(* CODESYS project Joint_7_TCP_new.project

Project tree, tasks and I/O mapping:
  Device : CODESYS Control arm CTH3 C37-000S1, 3S - Smart Software Solutions GmbH, version 3.5.4.30
    application Application
      libraries: Standard, * (System); Co-Trust Modbus Library, 1.1 (Co-Trust)
      task MainTask (cyclic, interval t#20ms, priority 1) calls Cyclic, TCP
      task EtherCAT_Master (cyclic, interval 2000 µs, priority 0) calls EtherCAT_Master.EtherCAT_Task [EtherCAT_Master.EtherCAT_Task], PLC_PRG
      program PLC_PRG [LD]
      global variables GVL
      trace Trace (task EtherCAT_Master): x.fSetPosition
      function block String_TO_HMI [ST]
      program Cyclic [LD]
      global variables PersistentVars
      program TCP [LD]
    SoftMotion General Axis Pool
    Co-trust LocalBus
    EtherCAT_Master : EtherCAT Master, 3S - Smart Software Solutions GmbH, version 3.5.4.0
        settings: MasterCycleTime = 2000; SlaveAutoRestart = True; NetworkName = 'eth1'; SelectNetworkByName = True; SrcAddress1 = 96; SrcAddress2 = 1856707308
      CiA402_Motor_Control_Device_6 : SOMANET CiA402 Drive, Synapticon GmbH, version Revision=16#0A000002
          settings: Number of Outputs = 7; Number of Inputs = 5; Number of Infos about Outputs = 7; Number of Infos about Inputs = 5; EnableExpertSettings = True; CheckProductID = False; CheckVendorID = False; Sync.Length = 19; Sync.Length = 13; FMMU.Length = 19; FMMU.Length = 13; DC enable = 1; DC sync0 enable = 1; DC sync0 shift time = 0; DC sync1 enable = 0; DC sync1 shift time = 0; DCSetting = 1; RxTxPdo.Sm = -1; RxTxPdo.Sm = -1; RxTxPdo.Sm = -1; RxTxPdo.Sm = -1; RxTxPdo.Sm = -1
          unmapped channels: Controlword, Op Mode, Target Torque, Target Position, Target Velocity, Torque offset, Tuning command, Statusword, Op Mode Display, Position Value, Velocity Value, Torque Value
        Joint_6 : SM_Drive_GenericDSP402, 3S - Smart Software Solutions GmbH, order no. 0, version 3.5.4.10
            settings: dwRatioTechUnitsDenom = 26214400; ScalingIncs = 262144; ScalingMotorTurns2 = 100; AdrOffset_8010 = 120; BitOffset_8010 = 0; BitLength_8010 = 16; Address_8010 = '%QW60'; Type_8010 = 'UINT'; AddressPointer_8010 = ADR(%QW60); AdrOffset_8020 = 128; BitOffset_8020 = 0; BitLength_8020 = 32; Address_8020 = '%QD32'; Type_8020 = 'DINT'; AddressPointer_8020 = ADR(%QD32); AdrOffset_8030 = 132; BitOffset_8030 = 0; BitLength_8030 = 32; Address_8030 = '%QD33'; Type_8030 = 'DINT'; AddressPointer_8030 = ADR(%QD33); AdrOffset_8040 = 124; BitOffset_8040 = 0; BitLength_8040 = 16; Address_8040 = '%QW62'; Type_8040 = 'INT'; AddressPointer_8040 = ADR(%QW62); AdrOffset_8050 = 122; BitOffset_8050 = 0; BitLength_8050 = 8; Address_8050 = '%QB122'; Type_8050 = 'SINT'; AddressPointer_8050 = ADR(%QB122); AdrOffset_8060 = 16#FFFFFFFF; BitOffset_8060 = 0; BitLength_8060 = 0; Address_8060 = ''; Type_8060 = ''; AddressPointer_8060 = 0; AdrOffset_8070 = 16#FFFFFFFF;
              BitOffset_8070 = 0; BitLength_8070 = 0; Address_8070 = ''; Type_8070 = ''; AddressPointer_8070 = 0; AdrOffset_8080 = 136; BitOffset_8080 = 0; BitLength_8080 = 16; Address_8080 = '%QW68'; Type_8080 = 'INT'; AddressPointer_8080 = ADR(%QW68); AdrOffset_8510 = 80; BitOffset_8510 = 0; BitLength_8510 = 16; Address_8510 = '%IW40'; Type_8510 = 'UINT'; AddressPointer_8510 = ADR(%IW40); AdrOffset_8520 = 84; BitOffset_8520 = 0; BitLength_8520 = 32; Address_8520 = '%ID21'; Type_8520 = 'DINT'; AddressPointer_8520 = ADR(%ID21); AdrOffset_8530 = 88; BitOffset_8530 = 0; BitLength_8530 = 32; Address_8530 = '%ID22'; Type_8530 = 'DINT'; AddressPointer_8530 = ADR(%ID22); AdrOffset_8540 = 92; BitOffset_8540 = 0; BitLength_8540 = 16; Address_8540 = '%IW46'; Type_8540 = 'INT'; AddressPointer_8540 = ADR(%IW46); AdrOffset_8550 = 82; BitOffset_8550 = 0; BitLength_8550 = 8; Address_8550 = '%IB82'; Type_8550 = 'SINT';
              AddressPointer_8550 = ADR(%IB82); AdrOffset_8560 = 16#FFFFFFFF; BitOffset_8560 = 0; BitLength_8560 = 0; Address_8560 = ''; Type_8560 = ''; AddressPointer_8560 = 0; AdrOffset_8570 = 16#FFFFFFFF; BitOffset_8570 = 0; BitLength_8570 = 0; Address_8570 = ''; Type_8570 = ''; AddressPointer_8570 = 0; AdrOffset_8580 = 16#FFFFFFFF; BitOffset_8580 = 0; BitLength_8580 = 0; Address_8580 = ''; Type_8580 = ''; AddressPointer_8580 = 0; AdrOffset_8590 = 16#FFFFFFFF; BitOffset_8590 = 0; BitLength_8590 = 0; Address_8590 = ''; Type_8590 = ''; AddressPointer_8590 = 0; AdrOffset_8600 = 16#FFFFFFFF; BitOffset_8600 = 0; BitLength_8600 = 0; Address_8600 = ''; Type_8600 = ''; AddressPointer_8600 = 0; AdrOffset_8600 = 16#FFFFFFFF; BitOffset_8600 = 0; BitLength_8600 = 0; Address_8610 = ''; Type_8610 = ''; AddressPointer_8610 = 0
      CiA402_Motor_Control_Device_4 : SOMANET CiA402 Drive, Synapticon GmbH, version Revision=16#0A000002
          settings: Number of Outputs = 7; Number of Inputs = 5; Number of Infos about Outputs = 7; Number of Infos about Inputs = 5; EnableExpertSettings = True; CheckProductID = False; CheckVendorID = False; Sync.Length = 19; Sync.Length = 13; FMMU.Length = 19; FMMU.Length = 13; DC enable = 1; DC sync0 enable = 1; DC sync0 shift time = 0; DC sync1 enable = 0; DC sync1 shift time = 0; DCSetting = 1; RxTxPdo.Sm = -1; RxTxPdo.Sm = -1; RxTxPdo.Sm = -1; RxTxPdo.Sm = -1; RxTxPdo.Sm = -1
          unmapped channels: Controlword, Op Mode, Target Torque, Target Position, Target Velocity, Torque offset, Tuning command, Statusword, Op Mode Display, Position Value, Velocity Value, Torque Value
        Joint_4 : SM_Drive_GenericDSP402, 3S - Smart Software Solutions GmbH, order no. 0, version 3.5.4.10
            settings: dwRatioTechUnitsDenom = 26214400; fSWLimitDeceleration = 0.0; fSWErrorMaxDistance = 0.0; ScalingIncs = 262144; ScalingMotorTurns2 = 100; AdrOffset_8010 = 72; BitOffset_8010 = 0; BitLength_8010 = 16; Address_8010 = '%QW36'; Type_8010 = 'UINT'; AddressPointer_8010 = ADR(%QW36); AdrOffset_8020 = 80; BitOffset_8020 = 0; BitLength_8020 = 32; Address_8020 = '%QD20'; Type_8020 = 'DINT'; AddressPointer_8020 = ADR(%QD20); AdrOffset_8030 = 84; BitOffset_8030 = 0; BitLength_8030 = 32; Address_8030 = '%QD21'; Type_8030 = 'DINT'; AddressPointer_8030 = ADR(%QD21); AdrOffset_8040 = 76; BitOffset_8040 = 0; BitLength_8040 = 16; Address_8040 = '%QW38'; Type_8040 = 'INT'; AddressPointer_8040 = ADR(%QW38); AdrOffset_8050 = 74; BitOffset_8050 = 0; BitLength_8050 = 8; Address_8050 = '%QB74'; Type_8050 = 'SINT'; AddressPointer_8050 = ADR(%QB74); AdrOffset_8060 = 16#FFFFFFFF; BitOffset_8060 = 0; BitLength_8060 = 0; Address_8060 = ''; Type_8060 = '';
              AddressPointer_8060 = 0; AdrOffset_8070 = 16#FFFFFFFF; BitOffset_8070 = 0; BitLength_8070 = 0; Address_8070 = ''; Type_8070 = ''; AddressPointer_8070 = 0; AdrOffset_8080 = 88; BitOffset_8080 = 0; BitLength_8080 = 16; Address_8080 = '%QW44'; Type_8080 = 'INT'; AddressPointer_8080 = ADR(%QW44); AdrOffset_8510 = 48; BitOffset_8510 = 0; BitLength_8510 = 16; Address_8510 = '%IW24'; Type_8510 = 'UINT'; AddressPointer_8510 = ADR(%IW24); AdrOffset_8520 = 52; BitOffset_8520 = 0; BitLength_8520 = 32; Address_8520 = '%ID13'; Type_8520 = 'DINT'; AddressPointer_8520 = ADR(%ID13); AdrOffset_8530 = 56; BitOffset_8530 = 0; BitLength_8530 = 32; Address_8530 = '%ID14'; Type_8530 = 'DINT'; AddressPointer_8530 = ADR(%ID14); AdrOffset_8540 = 60; BitOffset_8540 = 0; BitLength_8540 = 16; Address_8540 = '%IW30'; Type_8540 = 'INT'; AddressPointer_8540 = ADR(%IW30); AdrOffset_8550 = 50; BitOffset_8550 = 0; BitLength_8550 = 8;
              Address_8550 = '%IB50'; Type_8550 = 'SINT'; AddressPointer_8550 = ADR(%IB50); AdrOffset_8560 = 16#FFFFFFFF; BitOffset_8560 = 0; BitLength_8560 = 0; Address_8560 = ''; Type_8560 = ''; AddressPointer_8560 = 0; AdrOffset_8570 = 16#FFFFFFFF; BitOffset_8570 = 0; BitLength_8570 = 0; Address_8570 = ''; Type_8570 = ''; AddressPointer_8570 = 0; AdrOffset_8580 = 16#FFFFFFFF; BitOffset_8580 = 0; BitLength_8580 = 0; Address_8580 = ''; Type_8580 = ''; AddressPointer_8580 = 0; AdrOffset_8590 = 16#FFFFFFFF; BitOffset_8590 = 0; BitLength_8590 = 0; Address_8590 = ''; Type_8590 = ''; AddressPointer_8590 = 0; AdrOffset_8600 = 16#FFFFFFFF; BitOffset_8600 = 0; BitLength_8600 = 0; Address_8600 = ''; Type_8600 = ''; AddressPointer_8600 = 0; AdrOffset_8600 = 16#FFFFFFFF; BitOffset_8600 = 0; BitLength_8600 = 0; Address_8610 = ''; Type_8610 = ''; AddressPointer_8610 = 0
      CiA402_Motor_Control_Device_2 : SOMANET CiA402 Drive, Synapticon GmbH, version Revision=16#0A000002
          settings: Number of Outputs = 7; Number of Inputs = 5; Number of Infos about Outputs = 7; Number of Infos about Inputs = 5; EnableExpertSettings = True; CheckProductID = False; CheckVendorID = False; Sync.Length = 19; Sync.Length = 13; FMMU.Length = 19; FMMU.Length = 13; DC enable = 1; DC sync0 enable = 1; DC sync0 shift time = 0; DC sync1 enable = 0; DC sync1 shift time = 0; DCSetting = 1; RxTxPdo.Sm = -1; RxTxPdo.Sm = -1; RxTxPdo.Sm = -1; RxTxPdo.Sm = -1; RxTxPdo.Sm = -1
          unmapped channels: Controlword, Op Mode, Target Torque, Target Position, Target Velocity, Torque offset, Tuning command, Statusword, Op Mode Display, Position Value, Velocity Value, Torque Value
        Joint_2 : SM_Drive_GenericDSP402, 3S - Smart Software Solutions GmbH, order no. 0, version 3.5.4.10
            settings: dwRatioTechUnitsDenom = 31457280; ScalingIncs = 262144; ScalingMotorTurns2 = 120; AdrOffset_8010 = 24; BitOffset_8010 = 0; BitLength_8010 = 16; Address_8010 = '%QW12'; Type_8010 = 'UINT'; AddressPointer_8010 = ADR(%QW12); AdrOffset_8020 = 32; BitOffset_8020 = 0; BitLength_8020 = 32; Address_8020 = '%QD8'; Type_8020 = 'DINT'; AddressPointer_8020 = ADR(%QD8); AdrOffset_8030 = 36; BitOffset_8030 = 0; BitLength_8030 = 32; Address_8030 = '%QD9'; Type_8030 = 'DINT'; AddressPointer_8030 = ADR(%QD9); AdrOffset_8040 = 28; BitOffset_8040 = 0; BitLength_8040 = 16; Address_8040 = '%QW14'; Type_8040 = 'INT'; AddressPointer_8040 = ADR(%QW14); AdrOffset_8050 = 26; BitOffset_8050 = 0; BitLength_8050 = 8; Address_8050 = '%QB26'; Type_8050 = 'SINT'; AddressPointer_8050 = ADR(%QB26); AdrOffset_8060 = 16#FFFFFFFF; BitOffset_8060 = 0; BitLength_8060 = 0; Address_8060 = ''; Type_8060 = ''; AddressPointer_8060 = 0; AdrOffset_8070 = 16#FFFFFFFF;
              BitOffset_8070 = 0; BitLength_8070 = 0; Address_8070 = ''; Type_8070 = ''; AddressPointer_8070 = 0; AdrOffset_8080 = 40; BitOffset_8080 = 0; BitLength_8080 = 16; Address_8080 = '%QW20'; Type_8080 = 'INT'; AddressPointer_8080 = ADR(%QW20); AdrOffset_8510 = 16; BitOffset_8510 = 0; BitLength_8510 = 16; Address_8510 = '%IW8'; Type_8510 = 'UINT'; AddressPointer_8510 = ADR(%IW8); AdrOffset_8520 = 20; BitOffset_8520 = 0; BitLength_8520 = 32; Address_8520 = '%ID5'; Type_8520 = 'DINT'; AddressPointer_8520 = ADR(%ID5); AdrOffset_8530 = 24; BitOffset_8530 = 0; BitLength_8530 = 32; Address_8530 = '%ID6'; Type_8530 = 'DINT'; AddressPointer_8530 = ADR(%ID6); AdrOffset_8540 = 28; BitOffset_8540 = 0; BitLength_8540 = 16; Address_8540 = '%IW14'; Type_8540 = 'INT'; AddressPointer_8540 = ADR(%IW14); AdrOffset_8550 = 18; BitOffset_8550 = 0; BitLength_8550 = 8; Address_8550 = '%IB18'; Type_8550 = 'SINT';
              AddressPointer_8550 = ADR(%IB18); AdrOffset_8560 = 16#FFFFFFFF; BitOffset_8560 = 0; BitLength_8560 = 0; Address_8560 = ''; Type_8560 = ''; AddressPointer_8560 = 0; AdrOffset_8570 = 16#FFFFFFFF; BitOffset_8570 = 0; BitLength_8570 = 0; Address_8570 = ''; Type_8570 = ''; AddressPointer_8570 = 0; AdrOffset_8580 = 16#FFFFFFFF; BitOffset_8580 = 0; BitLength_8580 = 0; Address_8580 = ''; Type_8580 = ''; AddressPointer_8580 = 0; AdrOffset_8590 = 16#FFFFFFFF; BitOffset_8590 = 0; BitLength_8590 = 0; Address_8590 = ''; Type_8590 = ''; AddressPointer_8590 = 0; AdrOffset_8600 = 16#FFFFFFFF; BitOffset_8600 = 0; BitLength_8600 = 0; Address_8600 = ''; Type_8600 = ''; AddressPointer_8600 = 0; AdrOffset_8600 = 16#FFFFFFFF; BitOffset_8600 = 0; BitLength_8600 = 0; Address_8610 = ''; Type_8610 = ''; AddressPointer_8610 = 0
      CiA402_Motor_Control_Device : SOMANET CiA402 Drive, Synapticon GmbH, version Revision=16#0A000002
          settings: Number of Outputs = 7; Number of Inputs = 5; Number of Infos about Outputs = 7; Number of Infos about Inputs = 5; EnableExpertSettings = True; CheckProductID = False; CheckVendorID = False; Sync.Length = 19; Sync.Length = 13; FMMU.Length = 19; FMMU.Length = 13; DC enable = 1; DC sync0 enable = 1; DC sync0 shift time = 0; DC sync1 enable = 0; DC sync1 shift time = 0; DCSetting = 1; RxTxPdo.Sm = -1; RxTxPdo.Sm = -1; RxTxPdo.Sm = -1; RxTxPdo.Sm = -1; RxTxPdo.Sm = -1
          unmapped channels: Controlword, Op Mode, Target Torque, Target Position, Target Velocity, Torque offset, Tuning command, Statusword, Op Mode Display, Position Value, Velocity Value, Torque Value
        Joint_7 : SM_Drive_GenericDSP402, 3S - Smart Software Solutions GmbH, order no. 0, version 3.5.4.10
            settings: dwRatioTechUnitsDenom = 26214400; ScalingIncs = 262144; ScalingMotorTurns2 = 100; AdrOffset_8010 = 144; BitOffset_8010 = 0; BitLength_8010 = 16; Address_8010 = '%QW72'; Type_8010 = 'UINT'; AddressPointer_8010 = ADR(%QW72); AdrOffset_8020 = 152; BitOffset_8020 = 0; BitLength_8020 = 32; Address_8020 = '%QD38'; Type_8020 = 'DINT'; AddressPointer_8020 = ADR(%QD38); AdrOffset_8030 = 156; BitOffset_8030 = 0; BitLength_8030 = 32; Address_8030 = '%QD39'; Type_8030 = 'DINT'; AddressPointer_8030 = ADR(%QD39); AdrOffset_8040 = 148; BitOffset_8040 = 0; BitLength_8040 = 16; Address_8040 = '%QW74'; Type_8040 = 'INT'; AddressPointer_8040 = ADR(%QW74); AdrOffset_8050 = 146; BitOffset_8050 = 0; BitLength_8050 = 8; Address_8050 = '%QB146'; Type_8050 = 'SINT'; AddressPointer_8050 = ADR(%QB146); AdrOffset_8060 = 16#FFFFFFFF; BitOffset_8060 = 0; BitLength_8060 = 0; Address_8060 = ''; Type_8060 = ''; AddressPointer_8060 = 0; AdrOffset_8070 = 176;
              BitOffset_8070 = 0; BitLength_8070 = 32; Address_8070 = '%QD44'; Type_8070 = 'DINT'; AddressPointer_8070 = ADR(%QD44); AdrOffset_8080 = 160; BitOffset_8080 = 0; BitLength_8080 = 16; Address_8080 = '%QW80'; Type_8080 = 'INT'; AddressPointer_8080 = ADR(%QW80); AdrOffset_8510 = 96; BitOffset_8510 = 0; BitLength_8510 = 16; Address_8510 = '%IW48'; Type_8510 = 'UINT'; AddressPointer_8510 = ADR(%IW48); AdrOffset_8520 = 100; BitOffset_8520 = 0; BitLength_8520 = 32; Address_8520 = '%ID25'; Type_8520 = 'DINT'; AddressPointer_8520 = ADR(%ID25); AdrOffset_8530 = 104; BitOffset_8530 = 0; BitLength_8530 = 32; Address_8530 = '%ID26'; Type_8530 = 'DINT'; AddressPointer_8530 = ADR(%ID26); AdrOffset_8540 = 108; BitOffset_8540 = 0; BitLength_8540 = 16; Address_8540 = '%IW54'; Type_8540 = 'INT'; AddressPointer_8540 = ADR(%IW54); AdrOffset_8550 = 98; BitOffset_8550 = 0; BitLength_8550 = 8; Address_8550 = '%IB98'; Type_8550 = 'SINT';
              AddressPointer_8550 = ADR(%IB98); AdrOffset_8560 = 16#FFFFFFFF; BitOffset_8560 = 0; BitLength_8560 = 0; Address_8560 = ''; Type_8560 = ''; AddressPointer_8560 = 0; AdrOffset_8570 = 16#FFFFFFFF; BitOffset_8570 = 0; BitLength_8570 = 0; Address_8570 = ''; Type_8570 = ''; AddressPointer_8570 = 0; AdrOffset_8580 = 16#FFFFFFFF; BitOffset_8580 = 0; BitLength_8580 = 0; Address_8580 = ''; Type_8580 = ''; AddressPointer_8580 = 0; AdrOffset_8590 = 16#FFFFFFFF; BitOffset_8590 = 0; BitLength_8590 = 0; Address_8590 = ''; Type_8590 = ''; AddressPointer_8590 = 0; AdrOffset_8600 = 16#FFFFFFFF; BitOffset_8600 = 0; BitLength_8600 = 0; Address_8600 = ''; Type_8600 = ''; AddressPointer_8600 = 0; AdrOffset_8600 = 16#FFFFFFFF; BitOffset_8600 = 0; BitLength_8600 = 0; Address_8610 = ''; Type_8610 = ''; AddressPointer_8610 = 0; Automatic Mapping = FALSE
      CiA402_Motor_Control_Device_5 : SOMANET CiA402 Drive, Synapticon GmbH, version Revision=16#0A000002
          settings: Number of Outputs = 7; Number of Inputs = 5; Number of Infos about Outputs = 7; Number of Infos about Inputs = 5; EnableExpertSettings = True; CheckProductID = False; CheckVendorID = False; Sync.Length = 19; Sync.Length = 13; FMMU.Length = 19; FMMU.Length = 13; DC enable = 1; DC sync0 enable = 1; DC sync0 shift time = 0; DC sync1 enable = 0; DC sync1 shift time = 0; DCSetting = 1; RxTxPdo.Sm = -1; RxTxPdo.Sm = -1; RxTxPdo.Sm = -1; RxTxPdo.Sm = -1; RxTxPdo.Sm = -1
          unmapped channels: Controlword, Op Mode, Target Torque, Target Position, Target Velocity, Torque offset, Tuning command, Statusword, Op Mode Display, Position Value, Velocity Value, Torque Value
        Joint_5 : SM_Drive_GenericDSP402, 3S - Smart Software Solutions GmbH, order no. 0, version 3.5.4.10
            settings: dwRatioTechUnitsDenom = 26214400; ScalingIncs = 262144; ScalingMotorTurns2 = 100; AdrOffset_8010 = 96; BitOffset_8010 = 0; BitLength_8010 = 16; Address_8010 = '%QW48'; Type_8010 = 'UINT'; AddressPointer_8010 = ADR(%QW48); AdrOffset_8020 = 104; BitOffset_8020 = 0; BitLength_8020 = 32; Address_8020 = '%QD26'; Type_8020 = 'DINT'; AddressPointer_8020 = ADR(%QD26); AdrOffset_8030 = 108; BitOffset_8030 = 0; BitLength_8030 = 32; Address_8030 = '%QD27'; Type_8030 = 'DINT'; AddressPointer_8030 = ADR(%QD27); AdrOffset_8040 = 100; BitOffset_8040 = 0; BitLength_8040 = 16; Address_8040 = '%QW50'; Type_8040 = 'INT'; AddressPointer_8040 = ADR(%QW50); AdrOffset_8050 = 98; BitOffset_8050 = 0; BitLength_8050 = 8; Address_8050 = '%QB98'; Type_8050 = 'SINT'; AddressPointer_8050 = ADR(%QB98); AdrOffset_8060 = 16#FFFFFFFF; BitOffset_8060 = 0; BitLength_8060 = 0; Address_8060 = ''; Type_8060 = ''; AddressPointer_8060 = 0; AdrOffset_8070 = 16#FFFFFFFF;
              BitOffset_8070 = 0; BitLength_8070 = 0; Address_8070 = ''; Type_8070 = ''; AddressPointer_8070 = 0; AdrOffset_8080 = 112; BitOffset_8080 = 0; BitLength_8080 = 16; Address_8080 = '%QW56'; Type_8080 = 'INT'; AddressPointer_8080 = ADR(%QW56); AdrOffset_8510 = 64; BitOffset_8510 = 0; BitLength_8510 = 16; Address_8510 = '%IW32'; Type_8510 = 'UINT'; AddressPointer_8510 = ADR(%IW32); AdrOffset_8520 = 68; BitOffset_8520 = 0; BitLength_8520 = 32; Address_8520 = '%ID17'; Type_8520 = 'DINT'; AddressPointer_8520 = ADR(%ID17); AdrOffset_8530 = 72; BitOffset_8530 = 0; BitLength_8530 = 32; Address_8530 = '%ID18'; Type_8530 = 'DINT'; AddressPointer_8530 = ADR(%ID18); AdrOffset_8540 = 76; BitOffset_8540 = 0; BitLength_8540 = 16; Address_8540 = '%IW38'; Type_8540 = 'INT'; AddressPointer_8540 = ADR(%IW38); AdrOffset_8550 = 66; BitOffset_8550 = 0; BitLength_8550 = 8; Address_8550 = '%IB66'; Type_8550 = 'SINT';
              AddressPointer_8550 = ADR(%IB66); AdrOffset_8560 = 16#FFFFFFFF; BitOffset_8560 = 0; BitLength_8560 = 0; Address_8560 = ''; Type_8560 = ''; AddressPointer_8560 = 0; AdrOffset_8570 = 16#FFFFFFFF; BitOffset_8570 = 0; BitLength_8570 = 0; Address_8570 = ''; Type_8570 = ''; AddressPointer_8570 = 0; AdrOffset_8580 = 16#FFFFFFFF; BitOffset_8580 = 0; BitLength_8580 = 0; Address_8580 = ''; Type_8580 = ''; AddressPointer_8580 = 0; AdrOffset_8590 = 16#FFFFFFFF; BitOffset_8590 = 0; BitLength_8590 = 0; Address_8590 = ''; Type_8590 = ''; AddressPointer_8590 = 0; AdrOffset_8600 = 16#FFFFFFFF; BitOffset_8600 = 0; BitLength_8600 = 0; Address_8600 = ''; Type_8600 = ''; AddressPointer_8600 = 0; AdrOffset_8600 = 16#FFFFFFFF; BitOffset_8600 = 0; BitLength_8600 = 0; Address_8610 = ''; Type_8610 = ''; AddressPointer_8610 = 0
      CiA402_Motor_Control_Device_3 : SOMANET CiA402 Drive, Synapticon GmbH, version Revision=16#0A000002
          settings: Number of Outputs = 7; Number of Inputs = 5; Number of Infos about Outputs = 7; Number of Infos about Inputs = 5; EnableExpertSettings = True; CheckProductID = False; CheckVendorID = False; Sync.Length = 19; Sync.Length = 13; FMMU.Length = 19; FMMU.Length = 13; DC enable = 1; DC sync0 enable = 1; DC sync0 shift time = 0; DC sync1 enable = 0; DC sync1 shift time = 0; DCSetting = 1; RxTxPdo.Sm = -1; RxTxPdo.Sm = -1; RxTxPdo.Sm = -1; RxTxPdo.Sm = -1; RxTxPdo.Sm = -1
          unmapped channels: Controlword, Op Mode, Target Torque, Target Position, Target Velocity, Torque offset, Tuning command, Statusword, Op Mode Display, Position Value, Velocity Value, Torque Value
        Joint_3 : SM_Drive_GenericDSP402, 3S - Smart Software Solutions GmbH, order no. 0, version 3.5.4.10
            settings: dwRatioTechUnitsDenom = 31457280; ScalingIncs = 262144; ScalingMotorTurns2 = 120; AdrOffset_8010 = 48; BitOffset_8010 = 0; BitLength_8010 = 16; Address_8010 = '%QW24'; Type_8010 = 'UINT'; AddressPointer_8010 = ADR(%QW24); AdrOffset_8020 = 56; BitOffset_8020 = 0; BitLength_8020 = 32; Address_8020 = '%QD14'; Type_8020 = 'DINT'; AddressPointer_8020 = ADR(%QD14); AdrOffset_8030 = 60; BitOffset_8030 = 0; BitLength_8030 = 32; Address_8030 = '%QD15'; Type_8030 = 'DINT'; AddressPointer_8030 = ADR(%QD15); AdrOffset_8040 = 52; BitOffset_8040 = 0; BitLength_8040 = 16; Address_8040 = '%QW26'; Type_8040 = 'INT'; AddressPointer_8040 = ADR(%QW26); AdrOffset_8050 = 50; BitOffset_8050 = 0; BitLength_8050 = 8; Address_8050 = '%QB50'; Type_8050 = 'SINT'; AddressPointer_8050 = ADR(%QB50); AdrOffset_8060 = 16#FFFFFFFF; BitOffset_8060 = 0; BitLength_8060 = 0; Address_8060 = ''; Type_8060 = ''; AddressPointer_8060 = 0; AdrOffset_8070 = 16#FFFFFFFF;
              BitOffset_8070 = 0; BitLength_8070 = 0; Address_8070 = ''; Type_8070 = ''; AddressPointer_8070 = 0; AdrOffset_8080 = 64; BitOffset_8080 = 0; BitLength_8080 = 16; Address_8080 = '%QW32'; Type_8080 = 'INT'; AddressPointer_8080 = ADR(%QW32); AdrOffset_8510 = 32; BitOffset_8510 = 0; BitLength_8510 = 16; Address_8510 = '%IW16'; Type_8510 = 'UINT'; AddressPointer_8510 = ADR(%IW16); AdrOffset_8520 = 36; BitOffset_8520 = 0; BitLength_8520 = 32; Address_8520 = '%ID9'; Type_8520 = 'DINT'; AddressPointer_8520 = ADR(%ID9); AdrOffset_8530 = 40; BitOffset_8530 = 0; BitLength_8530 = 32; Address_8530 = '%ID10'; Type_8530 = 'DINT'; AddressPointer_8530 = ADR(%ID10); AdrOffset_8540 = 44; BitOffset_8540 = 0; BitLength_8540 = 16; Address_8540 = '%IW22'; Type_8540 = 'INT'; AddressPointer_8540 = ADR(%IW22); AdrOffset_8550 = 34; BitOffset_8550 = 0; BitLength_8550 = 8; Address_8550 = '%IB34'; Type_8550 = 'SINT';
              AddressPointer_8550 = ADR(%IB34); AdrOffset_8560 = 16#FFFFFFFF; BitOffset_8560 = 0; BitLength_8560 = 0; Address_8560 = ''; Type_8560 = ''; AddressPointer_8560 = 0; AdrOffset_8570 = 16#FFFFFFFF; BitOffset_8570 = 0; BitLength_8570 = 0; Address_8570 = ''; Type_8570 = ''; AddressPointer_8570 = 0; AdrOffset_8580 = 16#FFFFFFFF; BitOffset_8580 = 0; BitLength_8580 = 0; Address_8580 = ''; Type_8580 = ''; AddressPointer_8580 = 0; AdrOffset_8590 = 16#FFFFFFFF; BitOffset_8590 = 0; BitLength_8590 = 0; Address_8590 = ''; Type_8590 = ''; AddressPointer_8590 = 0; AdrOffset_8600 = 16#FFFFFFFF; BitOffset_8600 = 0; BitLength_8600 = 0; Address_8600 = ''; Type_8600 = ''; AddressPointer_8600 = 0; AdrOffset_8600 = 16#FFFFFFFF; BitOffset_8600 = 0; BitLength_8600 = 0; Address_8610 = ''; Type_8610 = ''; AddressPointer_8610 = 0
      CiA402_Motor_Control_Device_1 : SOMANET CiA402 Drive, Synapticon GmbH, version Revision=16#0A000002
          settings: Number of Outputs = 7; Number of Inputs = 5; Number of Infos about Outputs = 7; Number of Infos about Inputs = 5; EnableExpertSettings = True; CheckProductID = False; CheckVendorID = False; Sync.Length = 19; Sync.Length = 13; FMMU.Length = 19; FMMU.Length = 13; DC enable = 1; DC sync0 enable = 1; DC sync0 shift time = 0; DC sync1 enable = 0; DC sync1 shift time = 0; DCSetting = 1; RxTxPdo.Sm = -1; RxTxPdo.Sm = -1; RxTxPdo.Sm = -1; RxTxPdo.Sm = -1; RxTxPdo.Sm = -1
          unmapped channels: Controlword, Op Mode, Target Torque, Target Position, Target Velocity, Torque offset, Tuning command, Statusword, Op Mode Display, Position Value, Velocity Value, Torque Value
        Joint_1 : SM_Drive_GenericDSP402, 3S - Smart Software Solutions GmbH, order no. 0, version 3.5.4.10
            settings: dwRatioTechUnitsDenom = 31457280; ScalingIncs = 262144; ScalingMotorTurns2 = 120; AdrOffset_8010 = 0; BitOffset_8010 = 0; BitLength_8010 = 16; Address_8010 = '%QW0'; Type_8010 = 'UINT'; AddressPointer_8010 = ADR(%QW0); AdrOffset_8020 = 8; BitOffset_8020 = 0; BitLength_8020 = 32; Address_8020 = '%QD2'; Type_8020 = 'DINT'; AddressPointer_8020 = ADR(%QD2); AdrOffset_8030 = 12; BitOffset_8030 = 0; BitLength_8030 = 32; Address_8030 = '%QD3'; Type_8030 = 'DINT'; AddressPointer_8030 = ADR(%QD3); AdrOffset_8040 = 4; BitOffset_8040 = 0; BitLength_8040 = 16; Address_8040 = '%QW2'; Type_8040 = 'INT'; AddressPointer_8040 = ADR(%QW2); AdrOffset_8050 = 2; BitOffset_8050 = 0; BitLength_8050 = 8; Address_8050 = '%QB2'; Type_8050 = 'SINT'; AddressPointer_8050 = ADR(%QB2); AdrOffset_8060 = 16#FFFFFFFF; BitOffset_8060 = 0; BitLength_8060 = 0; Address_8060 = ''; Type_8060 = ''; AddressPointer_8060 = 0; AdrOffset_8070 = 16#FFFFFFFF;
              BitOffset_8070 = 0; BitLength_8070 = 0; Address_8070 = ''; Type_8070 = ''; AddressPointer_8070 = 0; AdrOffset_8080 = 16; BitOffset_8080 = 0; BitLength_8080 = 16; Address_8080 = '%QW8'; Type_8080 = 'INT'; AddressPointer_8080 = ADR(%QW8); AdrOffset_8510 = 0; BitOffset_8510 = 0; BitLength_8510 = 16; Address_8510 = '%IW0'; Type_8510 = 'UINT'; AddressPointer_8510 = ADR(%IW0); AdrOffset_8520 = 4; BitOffset_8520 = 0; BitLength_8520 = 32; Address_8520 = '%ID1'; Type_8520 = 'DINT'; AddressPointer_8520 = ADR(%ID1); AdrOffset_8530 = 8; BitOffset_8530 = 0; BitLength_8530 = 32; Address_8530 = '%ID2'; Type_8530 = 'DINT'; AddressPointer_8530 = ADR(%ID2); AdrOffset_8540 = 12; BitOffset_8540 = 0; BitLength_8540 = 16; Address_8540 = '%IW6'; Type_8540 = 'INT'; AddressPointer_8540 = ADR(%IW6); AdrOffset_8550 = 2; BitOffset_8550 = 0; BitLength_8550 = 8; Address_8550 = '%IB2'; Type_8550 = 'SINT';
              AddressPointer_8550 = ADR(%IB2); AdrOffset_8560 = 16#FFFFFFFF; BitOffset_8560 = 0; BitLength_8560 = 0; Address_8560 = ''; Type_8560 = ''; AddressPointer_8560 = 0; AdrOffset_8570 = 16#FFFFFFFF; BitOffset_8570 = 0; BitLength_8570 = 0; Address_8570 = ''; Type_8570 = ''; AddressPointer_8570 = 0; AdrOffset_8580 = 16#FFFFFFFF; BitOffset_8580 = 0; BitLength_8580 = 0; Address_8580 = ''; Type_8580 = ''; AddressPointer_8580 = 0; AdrOffset_8590 = 16#FFFFFFFF; BitOffset_8590 = 0; BitLength_8590 = 0; Address_8590 = ''; Type_8590 = ''; AddressPointer_8590 = 0; AdrOffset_8600 = 16#FFFFFFFF; BitOffset_8600 = 0; BitLength_8600 = 0; Address_8600 = ''; Type_8600 = ''; AddressPointer_8600 = 0; AdrOffset_8600 = 16#FFFFFFFF; BitOffset_8600 = 0; BitLength_8600 = 0; Address_8610 = ''; Type_8610 = ''; AddressPointer_8610 = 0
*)

// Device/Application/GVL
VAR_GLOBAL
	Done_1: BOOL;
	Done_2: BOOL;
	Done_3: BOOL;
	Done_4: BOOL;
	Done_5: BOOL;
	Done_6: BOOL;
	Done_7: BOOL;
	MC_Power_4: MC_Power;
	ERR_1: BOOL;
	ERR_2: BOOL;
	ERR_3: BOOL;
	ERR_4: BOOL;
	ERR_5: BOOL;
	ERR_6: BOOL;
	ERR_7: BOOL;
	ZERO_P1: LREAL;
	ZERO_P2: LREAL;
	ZERO_P3: LREAL;
	ZERO_P4: LREAL;
	ZERO_P5: LREAL;
	ZERO_P6: LREAL;
	ZERO_P7: LREAL;
	 // 反馈实际位置1 单位圈数
	POSITION_1: LREAL; 
	// 反馈实际位置2单位圈数
	POSITION_2: LREAL;
	// 反馈实际位置3 单位圈数
	POSITION_3: LREAL;
    // 反馈实际位置4单位圈数
	POSITION_4: LREAL;
	// 反馈实际位置5 单位圈数
	POSITION_5: LREAL;
	// 反馈实际位置6单位圈数
	POSITION_6: LREAL;
	// 反馈实际位置7单位圈数
	POSITION_7: LREAL;
	// 反馈实际度数1精度0.001度
END_VAR

// Device/Application/PersistentVars
VAR_GLOBAL PERSISTENT RETAIN
	// 持续变量生成的实例路径
	PLC_PRG.P1_ZERO: DWORD;
	// 持续变量生成的实例路径
	PLC_PRG.P2_ZERO: DWORD;
	// 持续变量生成的实例路径
	PLC_PRG.P3_ZERO: DWORD;
	// 持续变量生成的实例路径
	PLC_PRG.P4_ZERO: DWORD;
	// 持续变量生成的实例路径
	PLC_PRG.P5_ZERO: DWORD;
	// 持续变量生成的实例路径
	PLC_PRG.P6_ZERO: DWORD;
	// 持续变量生成的实例路径
	PLC_PRG.P7_ZERO: DWORD;
END_VAR

// Device/Application/Cyclic
PROGRAM Cyclic
VAR
	R_TRIG1: R_TRIG;
	R_TRIG2: R_TRIG;
	R_TRIG3: R_TRIG;
	R_TRIG4: R_TRIG;
	R_TRIG5: R_TRIG;
	R_TRIG6: R_TRIG;
	R_TRIG7: R_TRIG;
	R_TRIG8: R_TRIG;
	PP2: LREAL;
	// 实际度数2
	PP6: LREAL;
	// 实际度数3
	PP7: LREAL;
	// 实际度数4
	PP5: LREAL;
	// 实际度数5
	PP4: LREAL;
	// 实际度数6
	PP3: LREAL;
	// 实际度数7
	PP1: LREAL;
	
	PP1A: REAL;
	PP2A: REAL;
	PP3A: REAL;
	PP4A: REAL;
	PP5A: REAL;
	PP6A: REAL;
	PP7A: REAL;
	PP1B: DINT;
	PP2B: DINT;
	PP3B: DINT;
	PP4B: DINT;
	PP5B: DINT;
	PP6B: DINT;
	PP7B: DINT;
	PROTECK_1: BOOL;
	PROTECK_2: BOOL;
	PROTECK_3: BOOL;
	PROTECK_4: BOOL;
	PROTECK_5: BOOL;
	PROTECK_6: BOOL;
	PROTECK_7: BOOL;
	PP1E: DINT;
	PP1F: DINT;
	PP1G: DINT;
	PP2E: DINT;
	PP3E: DINT;
	PP4E: DINT;
	PP5E: DINT;
	PP6E: DINT;
	PP7E: DINT;
	PP7F: DINT;
	PP6F: DINT;
	PP5F: DINT;
	PP4F: DINT;
	PP3F: DINT;
	PP2F: DINT;
	PP2G: DINT;
	PP3G: DINT;
	PP4G: DINT;
	PP5G: DINT;
	PP6G: DINT;
	PP7G: DINT;
	dssf: BOOL;
	ssss: BOOL;
	TON_0: TON;
	TON_1: TON;
END_VAR
VAR // added by the converter: edge detectors and wires of the graphical bodies
    _w1, _w2, _w3, _w4, _w5, _w6, _w7, _w8, _w9, _w10, _w11, _w12, _w13, _w14, _w15, _w16 : BOOL;
END_VAR

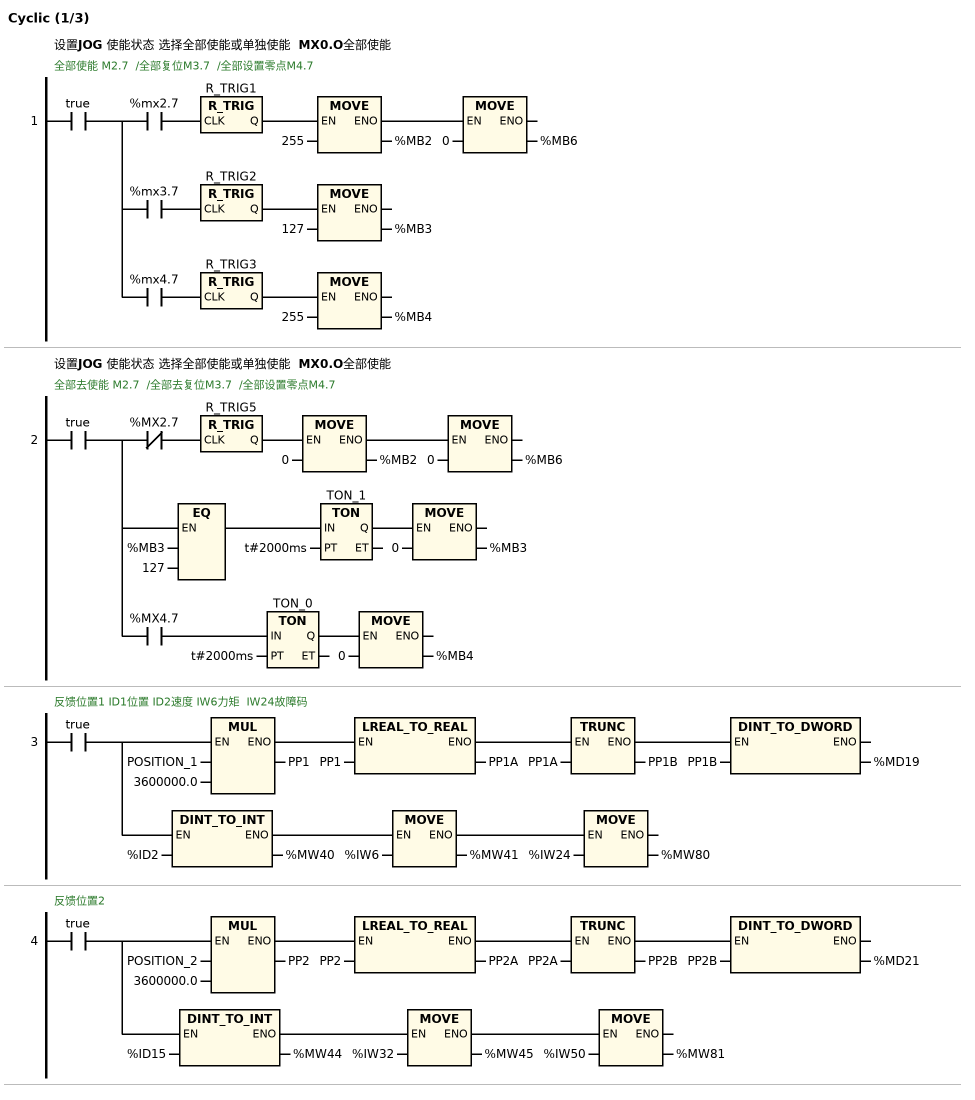
// NETWORK 1: 设置JOG 使能状态 选择全部使能或单独使能 MX0.O全部使能
// 全部使能 M2.7  /全部复位M3.7  /全部设置零点M4.7
R_TRIG1(CLK := true AND %mx2.7); // R_TRIG
_w1 := R_TRIG1.Q;
IF _w1 THEN %MB2 := 255; END_IF
IF _w1 THEN %MB6 := 0; END_IF
R_TRIG2(CLK := true AND %mx3.7); // R_TRIG
IF R_TRIG2.Q THEN %MB3 := 127; END_IF
R_TRIG3(CLK := true AND %mx4.7); // R_TRIG
IF R_TRIG3.Q THEN %MB4 := 255; END_IF

// NETWORK 2: 设置JOG 使能状态 选择全部使能或单独使能 MX0.O全部使能
// 全部去使能 M2.7  /全部去复位M3.7  /全部设置零点M4.7
R_TRIG5(CLK := true AND NOT %MX2.7); // R_TRIG
_w2 := R_TRIG5.Q;
IF _w2 THEN %MB2 := 0; END_IF
IF _w2 THEN %MB6 := 0; END_IF
TON_1(IN := true AND %MB3 = 127, PT := t#2000ms); // TON
IF TON_1.Q THEN %MB3 := 0; END_IF
TON_0(IN := true AND %MX4.7, PT := t#2000ms); // TON
IF TON_0.Q THEN %MB4 := 0; END_IF

// NETWORK 3
// 反馈位置1 ID1位置 ID2速度 IW6力矩  IW24故障码
//   POSITION_1: 反馈实际位置1 单位圈数
//   PP1: 实际度数7
_w3 := true;
IF _w3 THEN PP1 := POSITION_1 * 3600000.0; END_IF
IF _w3 THEN PP1A := LREAL_TO_REAL(PP1); END_IF
IF _w3 THEN PP1B := TRUNC(PP1A); END_IF
IF _w3 THEN %MD19 := DINT_TO_DWORD(PP1B); END_IF
_w4 := true;
IF _w4 THEN %MW40 := DINT_TO_INT(%ID2); END_IF
IF _w4 THEN %MW41 := %IW6; END_IF
IF _w4 THEN %MW80 := %IW24; END_IF

// NETWORK 4
// 反馈位置2
//   POSITION_2: 反馈实际位置2单位圈数
_w5 := true;
IF _w5 THEN PP2 := POSITION_2 * 3600000.0; END_IF
IF _w5 THEN PP2A := LREAL_TO_REAL(PP2); END_IF
IF _w5 THEN PP2B := TRUNC(PP2A); END_IF
IF _w5 THEN %MD21 := DINT_TO_DWORD(PP2B); END_IF
_w6 := true;
IF _w6 THEN %MW44 := DINT_TO_INT(%ID15); END_IF
IF _w6 THEN %MW45 := %IW32; END_IF
IF _w6 THEN %MW81 := %IW50; END_IF

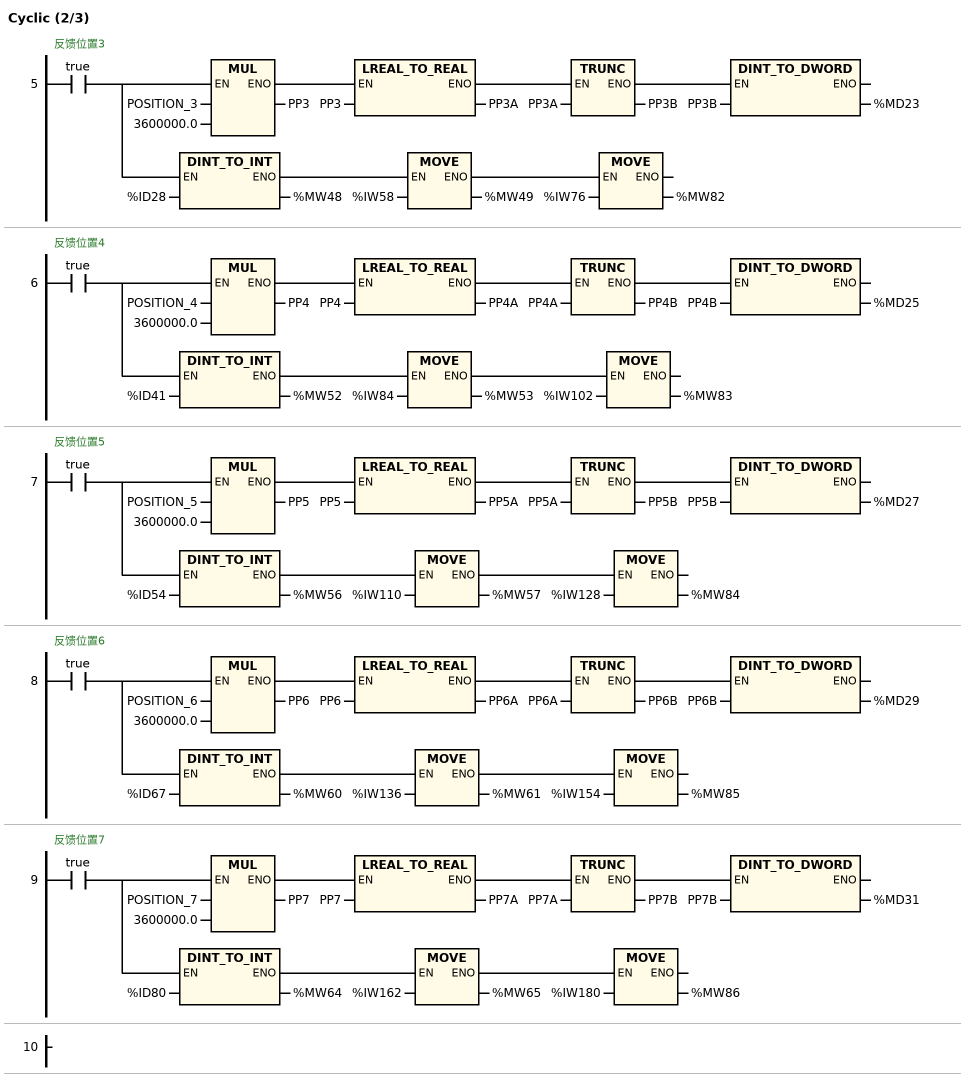
// NETWORK 5
// 反馈位置3
//   POSITION_3: 反馈实际位置3 单位圈数
//   PP3: 实际度数6
_w7 := true;
IF _w7 THEN PP3 := POSITION_3 * 3600000.0; END_IF
IF _w7 THEN PP3A := LREAL_TO_REAL(PP3); END_IF
IF _w7 THEN PP3B := TRUNC(PP3A); END_IF
IF _w7 THEN %MD23 := DINT_TO_DWORD(PP3B); END_IF
_w8 := true;
IF _w8 THEN %MW48 := DINT_TO_INT(%ID28); END_IF
IF _w8 THEN %MW49 := %IW58; END_IF
IF _w8 THEN %MW82 := %IW76; END_IF

// NETWORK 6
// 反馈位置4
//   POSITION_4: 反馈实际位置4单位圈数
//   PP4: 实际度数5
_w9 := true;
IF _w9 THEN PP4 := POSITION_4 * 3600000.0; END_IF
IF _w9 THEN PP4A := LREAL_TO_REAL(PP4); END_IF
IF _w9 THEN PP4B := TRUNC(PP4A); END_IF
IF _w9 THEN %MD25 := DINT_TO_DWORD(PP4B); END_IF
_w10 := true;
IF _w10 THEN %MW52 := DINT_TO_INT(%ID41); END_IF
IF _w10 THEN %MW53 := %IW84; END_IF
IF _w10 THEN %MW83 := %IW102; END_IF

// NETWORK 7
// 反馈位置5
//   POSITION_5: 反馈实际位置5 单位圈数
//   PP5: 实际度数4
_w11 := true;
IF _w11 THEN PP5 := POSITION_5 * 3600000.0; END_IF
IF _w11 THEN PP5A := LREAL_TO_REAL(PP5); END_IF
IF _w11 THEN PP5B := TRUNC(PP5A); END_IF
IF _w11 THEN %MD27 := DINT_TO_DWORD(PP5B); END_IF
_w12 := true;
IF _w12 THEN %MW56 := DINT_TO_INT(%ID54); END_IF
IF _w12 THEN %MW57 := %IW110; END_IF
IF _w12 THEN %MW84 := %IW128; END_IF

// NETWORK 8
// 反馈位置6
//   POSITION_6: 反馈实际位置6单位圈数
//   PP6: 实际度数2
_w13 := true;
IF _w13 THEN PP6 := POSITION_6 * 3600000.0; END_IF
IF _w13 THEN PP6A := LREAL_TO_REAL(PP6); END_IF
IF _w13 THEN PP6B := TRUNC(PP6A); END_IF
IF _w13 THEN %MD29 := DINT_TO_DWORD(PP6B); END_IF
_w14 := true;
IF _w14 THEN %MW60 := DINT_TO_INT(%ID67); END_IF
IF _w14 THEN %MW61 := %IW136; END_IF
IF _w14 THEN %MW85 := %IW154; END_IF

// NETWORK 9
// 反馈位置7
//   POSITION_7: 反馈实际位置7单位圈数
//   PP7: 实际度数3
_w15 := true;
IF _w15 THEN PP7 := POSITION_7 * 3600000.0; END_IF
IF _w15 THEN PP7A := LREAL_TO_REAL(PP7); END_IF
IF _w15 THEN PP7B := TRUNC(PP7A); END_IF
IF _w15 THEN %MD31 := DINT_TO_DWORD(PP7B); END_IF
_w16 := true;
IF _w16 THEN %MW64 := DINT_TO_INT(%ID80); END_IF
IF _w16 THEN %MW65 := %IW162; END_IF
IF _w16 THEN %MW86 := %IW180; END_IF

// NETWORK 10

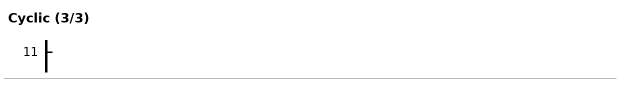
// NETWORK 11

END_PROGRAM

// Device/Application/TCP
PROGRAM TCP
VAR
	TT: POINTER TO WORD;
	MBUS_TCP_SLAVE_0: Co_Trust_Modbus_RTU_and_TCP.MBUS_TCP_SLAVE;
END_VAR

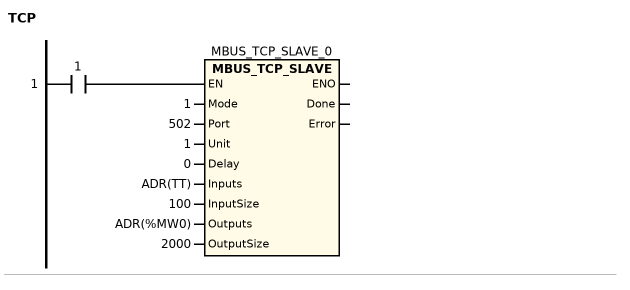
// NETWORK 1
IF 1 THEN
    MBUS_TCP_SLAVE_0(
        Mode := 1,
        Port := 502,
        Unit := 1,
        Delay := 0,
        Inputs := ADR(TT),
        InputSize := 100,
        Outputs := ADR(%MW0),
        OutputSize := 2000); // MBUS_TCP_SLAVE
END_IF

END_PROGRAM

// Device/Application/PLC_PRG
PROGRAM PLC_PRG
VAR
	MC_Power_0: MC_Power;
	MC_Power_1: MC_Power;
	MC_Power_2: MC_Power;
	MC_Power_3: MC_Power;
	MC_Power_5: MC_Power;
	MC_Power_6: MC_Power;
	MC_Power_7: MC_Power;
    MC_Reset_0: MC_Reset;
	MC_Reset_1: MC_Reset;
	MC_Reset_2: MC_Reset;
	MC_Reset_3: MC_Reset;
	MC_Reset_4: MC_Reset;
	MC_Reset_5: MC_Reset;
	MC_Reset_6: MC_Reset;
	MC_ReadActualPosition1: MC_ReadActualPosition;
	MC_ReadActualPosition2: MC_ReadActualPosition;
	MC_ReadActualPosition3: MC_ReadActualPosition;
	MC_ReadActualPosition4: MC_ReadActualPosition;
	MC_ReadActualPosition5: MC_ReadActualPosition;
	MC_ReadActualPosition6: MC_ReadActualPosition;
	MC_ReadActualPosition7: MC_ReadActualPosition;
	
	
	///////// （by MrRen-sdhm）  ////////////////
	
	INIT: BOOL := TRUE; // 初始化状态变量
	TON_INIT: TON; // 延时初始化触发器
	INIT_DONE: WORD := 1; // 控制器初始化成功
	
	// 目标位置-LREAL型(单位:度 10000倍)
	P1_LREAL: LREAL;
	P2_LREAL: LREAL;
	P3_LREAL: LREAL;
	P4_LREAL: LREAL;
	P5_LREAL: LREAL;
	P6_LREAL: LREAL;
	P7_LREAL: LREAL;
	
	// 目标位置-LREAL型(单位:转)
	P1_AIM: LREAL;
	P2_AIM: LREAL;
	P3_AIM: LREAL;
	P4_AIM: LREAL;
	P5_AIM: LREAL;
	P6_AIM: LREAL;
	P7_AIM: LREAL;	
	// 目标位置-DINT型(单位:度 10000倍)
	P1_DINT: DINT;	
	P2_DINT: DINT;	
	P3_DINT: DINT;
	P4_DINT: DINT;
	P5_DINT: DINT;
	P6_DINT: DINT;
	P7_DINT: DINT;

	R_TRIG_ZERO: R_TRIG;
	R_TRIG_RESET1: R_TRIG;
	R_TRIG_RESET2: R_TRIG;
	R_TRIG_RESET3: R_TRIG;
	R_TRIG_RESET4: R_TRIG;
	R_TRIG_RESET5: R_TRIG;
	R_TRIG_RESET6: R_TRIG;
	R_TRIG_RESET7: R_TRIG;
	
	// MC_MoveAbsolute相关
	MOVE_FLAG: BOOL; // MC_MoveAbsolute触发标志
	FLAG: BOOL := FALSE; // 脉冲发生器切换标志
	TP_1: TP;
	TP_2: TP;
	VELOCITY: LREAL := 1.0; // 速度 0.5
	ACCELERATION: LREAL := 1.0; // 加速度 0.15
	MC_MoveAbsolute_1: MC_MoveAbsolute;
	MC_MoveAbsolute_2: MC_MoveAbsolute;
	MC_MoveAbsolute_3: MC_MoveAbsolute;
	MC_MoveAbsolute_4: MC_MoveAbsolute;
	MC_MoveAbsolute_5: MC_MoveAbsolute;
	MC_MoveAbsolute_6: MC_MoveAbsolute;
	MC_MoveAbsolute_7: MC_MoveAbsolute;
	
	Back_Home: Bool := False;
END_VAR

VAR RETAIN PERSISTENT
	// 零位设为持续性变量保存
	P1_ZERO: DWORD;
	P2_ZERO: DWORD;
	P3_ZERO: DWORD;
	P4_ZERO: DWORD;
	P5_ZERO: DWORD;
	P6_ZERO: DWORD;
	P7_ZERO: DWORD;
END_VAR
VAR // added by the converter: edge detectors and wires of the graphical bodies
    _w1, _w2, _w3, _w4, _w5, _w6, _w7, _w8, _w9, _w10, _w11 : BOOL;
    _ft1 : F_TRIG;
END_VAR

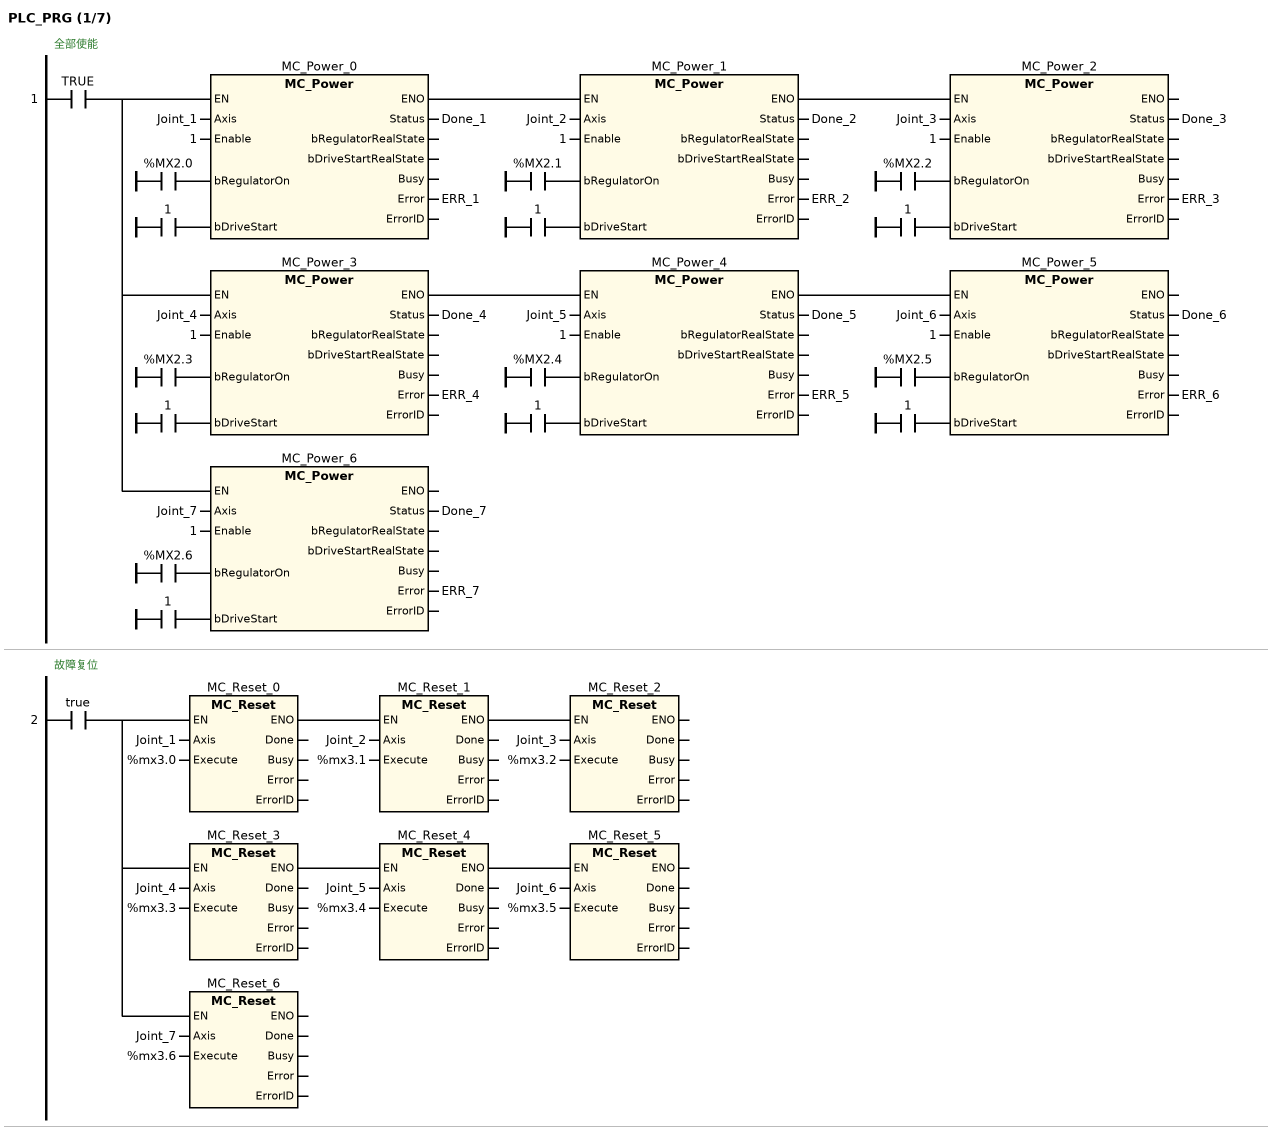
// NETWORK 1
// 全部使能
MC_Power_0(
    Axis := Joint_1,
    Enable := 1,
    bRegulatorOn := %MX2.0,
    bDriveStart := 1,
    Status => Done_1,
    Error => ERR_1); // MC_Power
MC_Power_1(
    Axis := Joint_2,
    Enable := 1,
    bRegulatorOn := %MX2.1,
    bDriveStart := 1,
    Status => Done_2,
    Error => ERR_2); // MC_Power
MC_Power_2(
    Axis := Joint_3,
    Enable := 1,
    bRegulatorOn := %MX2.2,
    bDriveStart := 1,
    Status => Done_3,
    Error => ERR_3); // MC_Power
MC_Power_3(
    Axis := Joint_4,
    Enable := 1,
    bRegulatorOn := %MX2.3,
    bDriveStart := 1,
    Status => Done_4,
    Error => ERR_4); // MC_Power
MC_Power_4(
    Axis := Joint_5,
    Enable := 1,
    bRegulatorOn := %MX2.4,
    bDriveStart := 1,
    Status => Done_5,
    Error => ERR_5); // MC_Power
MC_Power_5(
    Axis := Joint_6,
    Enable := 1,
    bRegulatorOn := %MX2.5,
    bDriveStart := 1,
    Status => Done_6,
    Error => ERR_6); // MC_Power
MC_Power_6(
    Axis := Joint_7,
    Enable := 1,
    bRegulatorOn := %MX2.6,
    bDriveStart := 1,
    Status => Done_7,
    Error => ERR_7); // MC_Power

// NETWORK 2
// 故障复位
_w1 := true;
IF _w1 THEN
    MC_Reset_0(Axis := Joint_1, Execute := %mx3.0); // MC_Reset
END_IF
IF _w1 THEN
    MC_Reset_1(Axis := Joint_2, Execute := %mx3.1); // MC_Reset
END_IF
IF _w1 THEN
    MC_Reset_2(Axis := Joint_3, Execute := %mx3.2); // MC_Reset
END_IF
_w2 := true;
IF _w2 THEN
    MC_Reset_3(Axis := Joint_4, Execute := %mx3.3); // MC_Reset
END_IF
IF _w2 THEN
    MC_Reset_4(Axis := Joint_5, Execute := %mx3.4); // MC_Reset
END_IF
IF _w2 THEN
    MC_Reset_5(Axis := Joint_6, Execute := %mx3.5); // MC_Reset
END_IF
IF true THEN
    MC_Reset_6(Axis := Joint_7, Execute := %mx3.6); // MC_Reset
END_IF

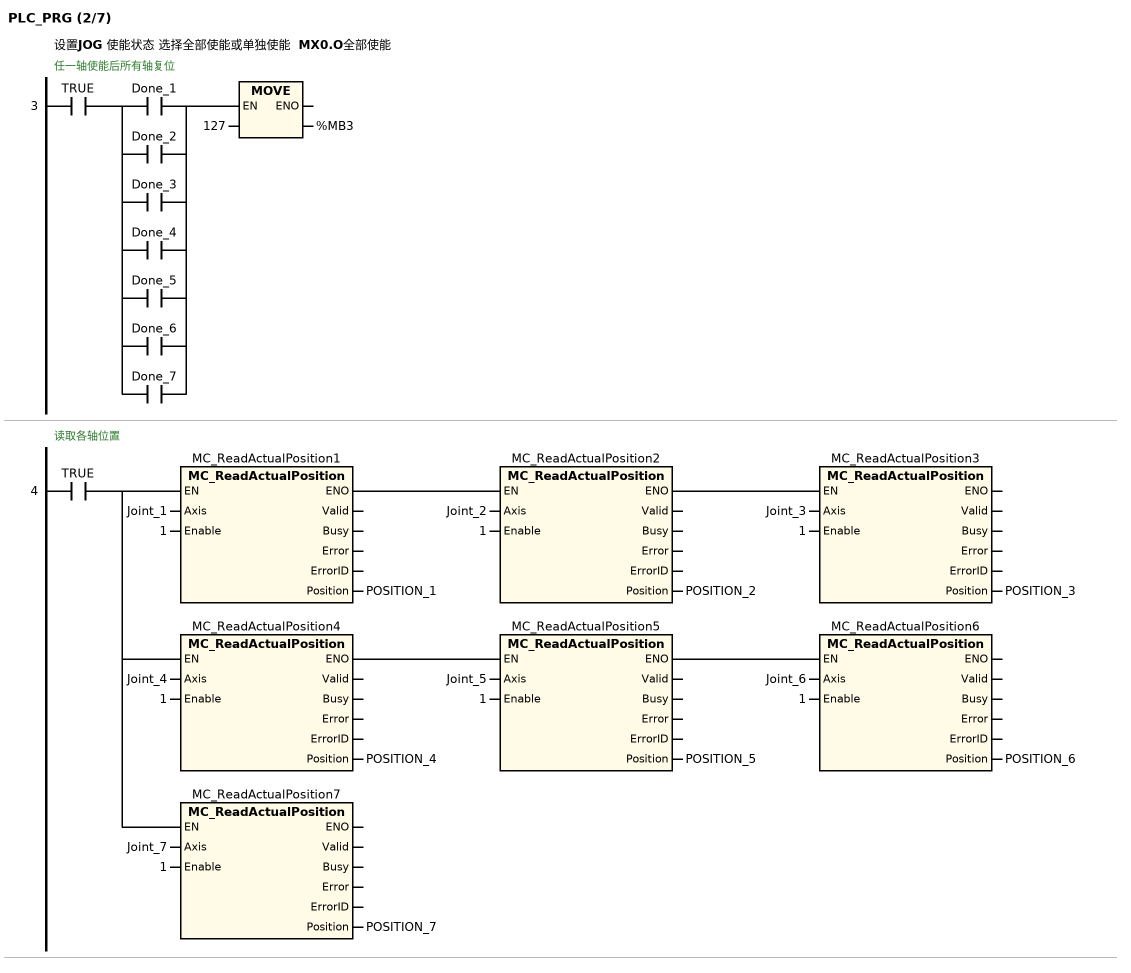
// NETWORK 3: 设置JOG 使能状态 选择全部使能或单独使能 MX0.O全部使能
// 任一轴使能后所有轴复位
IF TRUE AND (Done_1 OR Done_2 OR Done_3 OR Done_4 OR Done_5 OR Done_6 OR Done_7) THEN %MB3 := 127; END_IF

// NETWORK 4
// 读取各轴位置
//   POSITION_1: 反馈实际位置1 单位圈数
//   POSITION_2: 反馈实际位置2单位圈数
//   POSITION_3: 反馈实际位置3 单位圈数
//   POSITION_4: 反馈实际位置4单位圈数
//   POSITION_5: 反馈实际位置5 单位圈数
//   POSITION_6: 反馈实际位置6单位圈数
//   POSITION_7: 反馈实际位置7单位圈数
MC_ReadActualPosition1(Axis := Joint_1, Enable := 1, Position => POSITION_1); // MC_ReadActualPosition
MC_ReadActualPosition2(Axis := Joint_2, Enable := 1, Position => POSITION_2); // MC_ReadActualPosition
MC_ReadActualPosition3(Axis := Joint_3, Enable := 1, Position => POSITION_3); // MC_ReadActualPosition
MC_ReadActualPosition4(Axis := Joint_4, Enable := 1, Position => POSITION_4); // MC_ReadActualPosition
MC_ReadActualPosition5(Axis := Joint_5, Enable := 1, Position => POSITION_5); // MC_ReadActualPosition
MC_ReadActualPosition6(Axis := Joint_6, Enable := 1, Position => POSITION_6); // MC_ReadActualPosition
MC_ReadActualPosition7(Axis := Joint_7, Enable := 1, Position => POSITION_7); // MC_ReadActualPosition

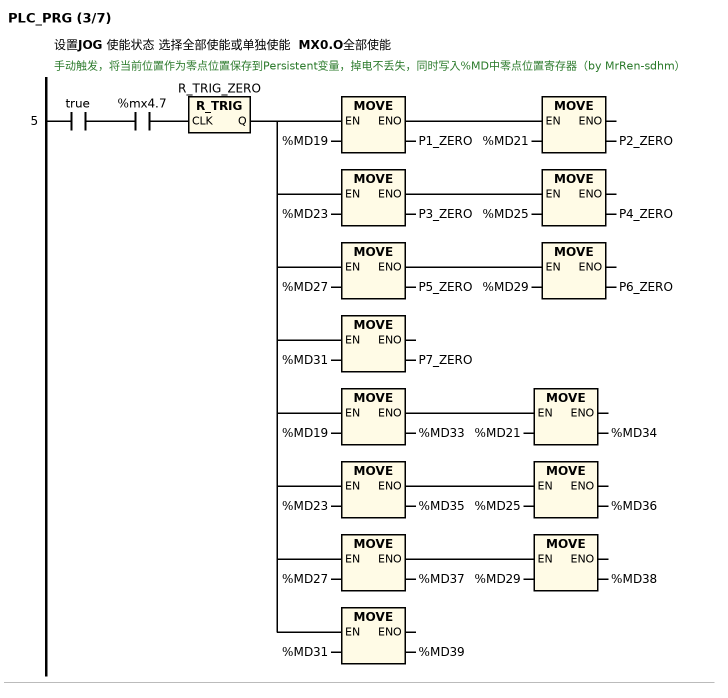
// NETWORK 5: 设置JOG 使能状态 选择全部使能或单独使能 MX0.O全部使能
// 手动触发，将当前位置作为零点位置保存到Persistent变量，掉电不丢失，同时写入%MD中零点位置寄存器（by MrRen-sdhm）
//   P1_ZERO: 零位设为持续性变量保存
R_TRIG_ZERO(CLK := true AND %mx4.7); // R_TRIG
_w3 := R_TRIG_ZERO.Q;
IF _w3 THEN P1_ZERO := %MD19; END_IF
IF _w3 THEN P2_ZERO := %MD21; END_IF
_w4 := R_TRIG_ZERO.Q;
IF _w4 THEN P3_ZERO := %MD23; END_IF
IF _w4 THEN P4_ZERO := %MD25; END_IF
_w5 := R_TRIG_ZERO.Q;
IF _w5 THEN P5_ZERO := %MD27; END_IF
IF _w5 THEN P6_ZERO := %MD29; END_IF
IF R_TRIG_ZERO.Q THEN P7_ZERO := %MD31; END_IF
_w6 := R_TRIG_ZERO.Q;
IF _w6 THEN %MD33 := %MD19; END_IF
IF _w6 THEN %MD34 := %MD21; END_IF
_w7 := R_TRIG_ZERO.Q;
IF _w7 THEN %MD35 := %MD23; END_IF
IF _w7 THEN %MD36 := %MD25; END_IF
_w8 := R_TRIG_ZERO.Q;
IF _w8 THEN %MD37 := %MD27; END_IF
IF _w8 THEN %MD38 := %MD29; END_IF
IF R_TRIG_ZERO.Q THEN %MD39 := %MD31; END_IF

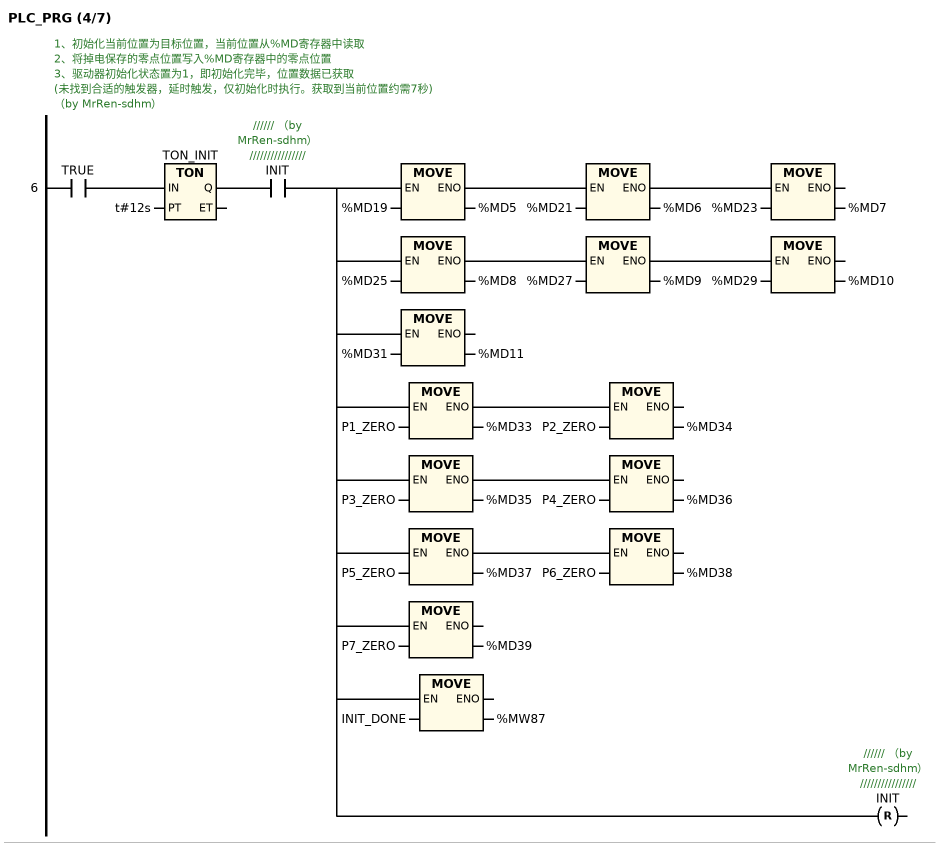
// NETWORK 6
// 1、初始化当前位置为目标位置，当前位置从%MD寄存器中读取
// 2、将掉电保存的零点位置写入%MD寄存器中的零点位置
// 3、驱动器初始化状态置为1，即初始化完毕，位置数据已获取
// (未找到合适的触发器，延时触发，仅初始化时执行。获取到当前位置约需7秒)
// （by MrRen-sdhm）
//   TON_INIT: 延时初始化触发器
//   INIT: ////// （by MrRen-sdhm） ////////////////
//   P1_ZERO: 零位设为持续性变量保存
//   INIT_DONE: 控制器初始化成功
TON_INIT(IN := TRUE, PT := t#12s); // TON
_w9 := TON_INIT.Q AND INIT;
IF _w9 THEN %MD5 := %MD19; END_IF
IF _w9 THEN %MD6 := %MD21; END_IF
IF _w9 THEN %MD7 := %MD23; END_IF
IF _w9 THEN %MD8 := %MD25; END_IF
IF _w9 THEN %MD9 := %MD27; END_IF
IF _w9 THEN %MD10 := %MD29; END_IF
IF _w9 THEN %MD11 := %MD31; END_IF
IF _w9 THEN %MD33 := P1_ZERO; END_IF
IF _w9 THEN %MD34 := P2_ZERO; END_IF
IF _w9 THEN %MD35 := P3_ZERO; END_IF
IF _w9 THEN %MD36 := P4_ZERO; END_IF
IF _w9 THEN %MD37 := P5_ZERO; END_IF
IF _w9 THEN %MD38 := P6_ZERO; END_IF
IF _w9 THEN %MD39 := P7_ZERO; END_IF
IF _w9 THEN %MW87 := INIT_DONE; END_IF
INIT R= _w9;

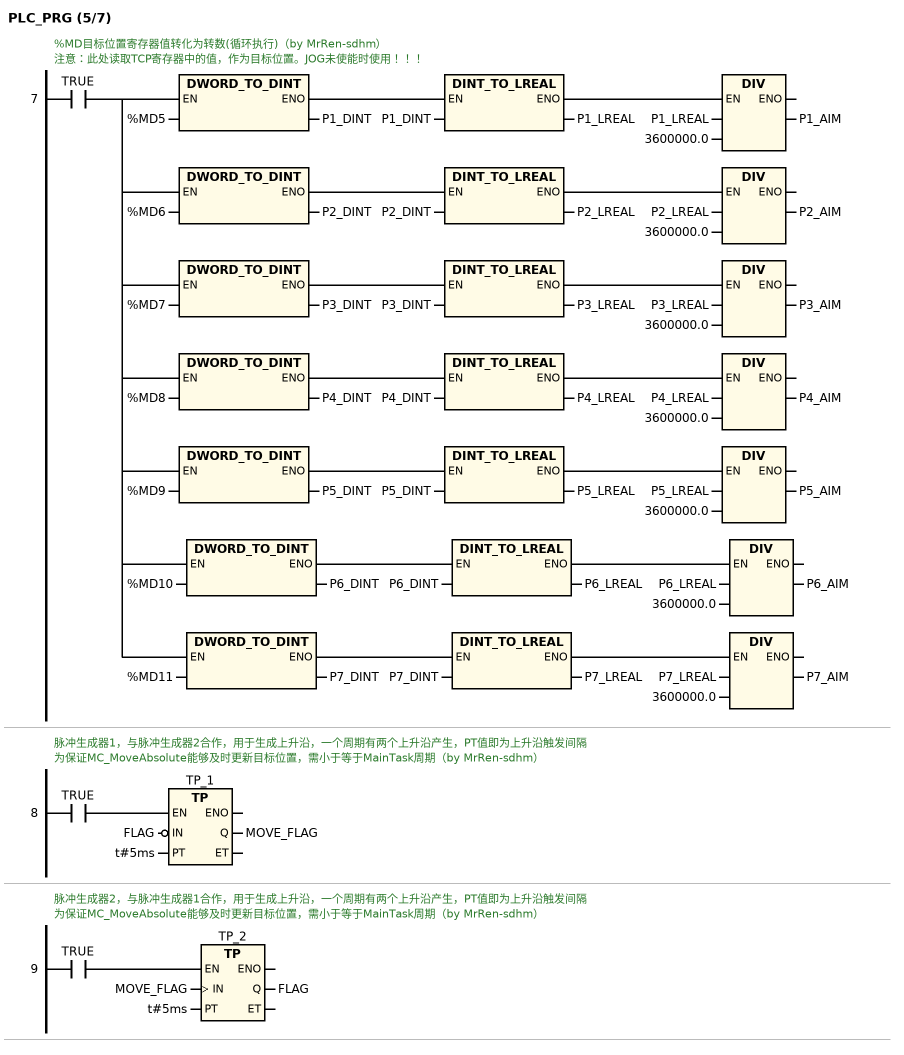
// NETWORK 7
// %MD目标位置寄存器值转化为转数(循环执行)（by MrRen-sdhm）
// 注意：此处读取TCP寄存器中的值，作为目标位置。JOG未使能时使用！！！
//   P1_DINT: 目标位置-DINT型(单位:度 10000倍)
//   P1_LREAL: 目标位置-LREAL型(单位:度 10000倍)
//   P1_AIM: 目标位置-LREAL型(单位:转)
P1_DINT := DWORD_TO_DINT(%MD5);
P1_LREAL := DINT_TO_LREAL(P1_DINT);
P1_AIM := P1_LREAL / 3600000.0;
P2_DINT := DWORD_TO_DINT(%MD6);
P2_LREAL := DINT_TO_LREAL(P2_DINT);
P2_AIM := P2_LREAL / 3600000.0;
P3_DINT := DWORD_TO_DINT(%MD7);
P3_LREAL := DINT_TO_LREAL(P3_DINT);
P3_AIM := P3_LREAL / 3600000.0;
P4_DINT := DWORD_TO_DINT(%MD8);
P4_LREAL := DINT_TO_LREAL(P4_DINT);
P4_AIM := P4_LREAL / 3600000.0;
P5_DINT := DWORD_TO_DINT(%MD9);
P5_LREAL := DINT_TO_LREAL(P5_DINT);
P5_AIM := P5_LREAL / 3600000.0;
P6_DINT := DWORD_TO_DINT(%MD10);
P6_LREAL := DINT_TO_LREAL(P6_DINT);
P6_AIM := P6_LREAL / 3600000.0;
P7_DINT := DWORD_TO_DINT(%MD11);
P7_LREAL := DINT_TO_LREAL(P7_DINT);
P7_AIM := P7_LREAL / 3600000.0;

// NETWORK 8
// 脉冲生成器1，与脉冲生成器2合作，用于生成上升沿，一个周期有两个上升沿产生，PT值即为上升沿触发间隔
// 为保证MC_MoveAbsolute能够及时更新目标位置，需小于等于MainTask周期（by MrRen-sdhm）
//   FLAG: 脉冲发生器切换标志
//   MOVE_FLAG: MC_MoveAbsolute触发标志
TP_1(IN := NOT FLAG, PT := t#5ms, Q => MOVE_FLAG); // TP

// NETWORK 9
// 脉冲生成器2，与脉冲生成器1合作，用于生成上升沿，一个周期有两个上升沿产生，PT值即为上升沿触发间隔
// 为保证MC_MoveAbsolute能够及时更新目标位置，需小于等于MainTask周期（by MrRen-sdhm）
//   MOVE_FLAG: MC_MoveAbsolute触发标志
//   FLAG: 脉冲发生器切换标志
_ft1(CLK := MOVE_FLAG);
TP_2(IN := _ft1.Q, PT := t#5ms, Q => FLAG); // TP

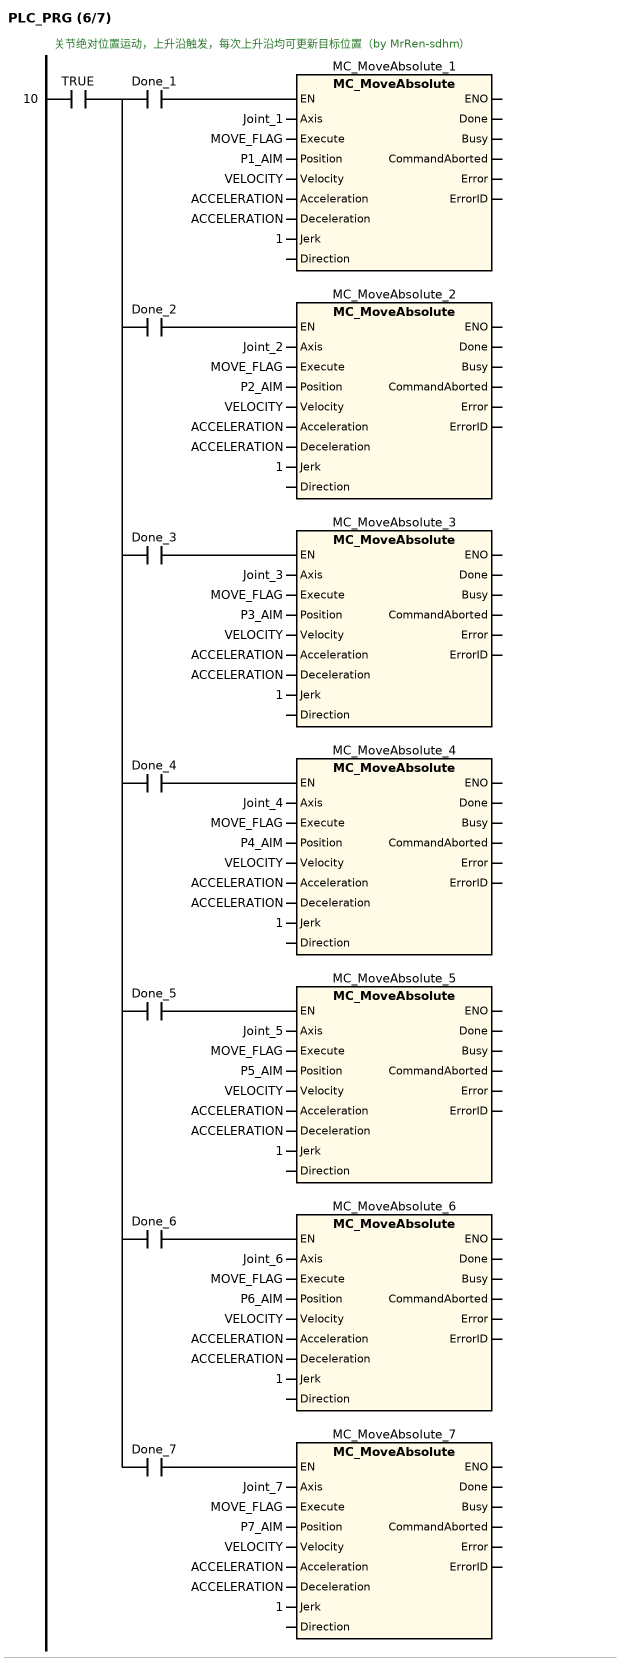
// NETWORK 10
// 关节绝对位置运动，上升沿触发，每次上升沿均可更新目标位置（by MrRen-sdhm）
//   MOVE_FLAG: MC_MoveAbsolute触发标志
//   P1_AIM: 目标位置-LREAL型(单位:转)
//   VELOCITY: 速度 0.5
//   ACCELERATION: 加速度 0.15
IF TRUE AND Done_1 THEN
    MC_MoveAbsolute_1(
        Axis := Joint_1,
        Execute := MOVE_FLAG,
        Position := P1_AIM,
        Velocity := VELOCITY,
        Acceleration := ACCELERATION,
        Deceleration := ACCELERATION,
        Jerk := 1); // MC_MoveAbsolute
END_IF
IF TRUE AND Done_2 THEN
    MC_MoveAbsolute_2(
        Axis := Joint_2,
        Execute := MOVE_FLAG,
        Position := P2_AIM,
        Velocity := VELOCITY,
        Acceleration := ACCELERATION,
        Deceleration := ACCELERATION,
        Jerk := 1); // MC_MoveAbsolute
END_IF
IF TRUE AND Done_3 THEN
    MC_MoveAbsolute_3(
        Axis := Joint_3,
        Execute := MOVE_FLAG,
        Position := P3_AIM,
        Velocity := VELOCITY,
        Acceleration := ACCELERATION,
        Deceleration := ACCELERATION,
        Jerk := 1); // MC_MoveAbsolute
END_IF
IF TRUE AND Done_4 THEN
    MC_MoveAbsolute_4(
        Axis := Joint_4,
        Execute := MOVE_FLAG,
        Position := P4_AIM,
        Velocity := VELOCITY,
        Acceleration := ACCELERATION,
        Deceleration := ACCELERATION,
        Jerk := 1); // MC_MoveAbsolute
END_IF
IF TRUE AND Done_5 THEN
    MC_MoveAbsolute_5(
        Axis := Joint_5,
        Execute := MOVE_FLAG,
        Position := P5_AIM,
        Velocity := VELOCITY,
        Acceleration := ACCELERATION,
        Deceleration := ACCELERATION,
        Jerk := 1); // MC_MoveAbsolute
END_IF
IF TRUE AND Done_6 THEN
    MC_MoveAbsolute_6(
        Axis := Joint_6,
        Execute := MOVE_FLAG,
        Position := P6_AIM,
        Velocity := VELOCITY,
        Acceleration := ACCELERATION,
        Deceleration := ACCELERATION,
        Jerk := 1); // MC_MoveAbsolute
END_IF
IF TRUE AND Done_7 THEN
    MC_MoveAbsolute_7(
        Axis := Joint_7,
        Execute := MOVE_FLAG,
        Position := P7_AIM,
        Velocity := VELOCITY,
        Acceleration := ACCELERATION,
        Deceleration := ACCELERATION,
        Jerk := 1); // MC_MoveAbsolute
END_IF

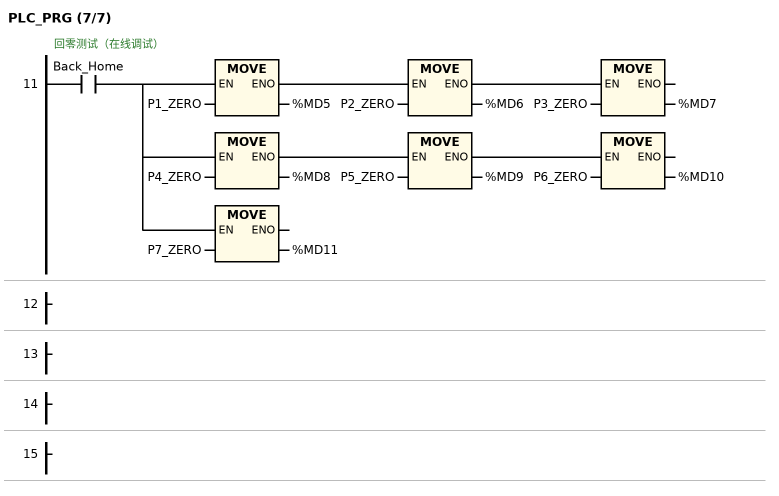
// NETWORK 11
// 回零测试（在线调试）
//   P1_ZERO: 零位设为持续性变量保存
_w10 := Back_Home;
IF _w10 THEN %MD5 := P1_ZERO; END_IF
IF _w10 THEN %MD6 := P2_ZERO; END_IF
IF _w10 THEN %MD7 := P3_ZERO; END_IF
_w11 := Back_Home;
IF _w11 THEN %MD8 := P4_ZERO; END_IF
IF _w11 THEN %MD9 := P5_ZERO; END_IF
IF _w11 THEN %MD10 := P6_ZERO; END_IF
IF Back_Home THEN %MD11 := P7_ZERO; END_IF

// NETWORK 12

// NETWORK 13

// NETWORK 14

// NETWORK 15

END_PROGRAM

// Device/Application/String_TO_HMI
FUNCTION_BLOCK String_TO_HMI
VAR_INPUT
	Stringin: STRING;
END_VAR
VAR_OUTPUT
	StringTOHmiout: STRING(80);
END_VAR
VAR
	Stringlen: INT;
	Oddchonse: INT;
	HalfStringlen: INT;
	Stringlenreal: REAL;
	Oddaddone: INT;
	OddString: STRING;
	OddStringDel: STRING;
	OddHalfStringlen: INT;
	EvenHalfStringlen: INT;
	Evenchonse: INT;
	EvenStringDel: STRING(255);
	EvenString: STRING(255);
	Stringchonse: INT;
	EmptyString: STRING(255);
	InsEvenStringchonse: INT;
	InsOddHalfStringlen: INT;
	InsEvenString: STRING;
	VarSTRING1: STRING(255);
	InsStringchonse: INT;
	InsOddString: STRING(255);
	IntegrationString: STRING(255);
	Insnum: INT;
	
	HalfSTringlenadd1: INT;
	Stringlen1: INT;
	STR_OUT: STRING;
	InsStringlen1: INT;
	straddlen: INT;
	stradd: STRING;
	straddout: STRING(255);
	RStringin: STRING;
	//Clearadd: INT;
END_VAR


   IF Stringin<>RStringin THEN

Stringlen:= LEN (Stringin);

HalfStringlen:=Stringlen/2;
Oddaddone:= Stringlen MOD 2;
IF Stringlen>1 THEN


//奇数处理
IF Oddaddone=1 THEN
OddHalfStringlen:=Stringlen/2+1;
END_IF
IF Oddaddone=0 THEN
OddHalfStringlen:=Stringlen/2;	
END_IF
FOR Oddchonse:=1 TO OddHalfStringlen  BY 1 DO
IF Oddchonse=1 AND OddHalfStringlen=1 THEN
OddStringDel:=  DELETE (Stringin,1,2);
END_IF
IF Oddchonse=2 AND OddHalfStringlen<>1 THEN
OddStringDel:=  DELETE (Stringin,1,Oddchonse); 
END_IF
IF Oddchonse>2 THEN
OddStringDel:= DELETE (OddStringDel,1,Oddchonse);	
END_IF	
END_FOR
OddString:=OddStringDel;	





//偶数处理
EvenHalfStringlen:=Stringlen/2;
FOR Evenchonse:=1 TO OddHalfStringlen BY 1 DO
IF Evenchonse=1 THEN
EvenStringDel := DELETE (Stringin,1,Evenchonse);
END_IF
IF Evenchonse>1 THEN
EvenStringDel := DELETE (EvenStringDel,1,Evenchonse);
END_IF	
END_FOR
IF Oddaddone=1 THEN
EvenString := CONCAT (EvenStringDel,' '); 
END_IF
IF Oddaddone=0 THEN
EvenString:=EvenStringDel;	
END_IF




//奇数偶数整合
FOR InsStringchonse:=1 TO OddHalfStringlen BY 1 DO
  InsOddString:= MID (OddString,1,InsStringchonse);
  IF InsStringchonse=1 THEN
    IntegrationString:= INSERT (EvenString,InsOddString,InsStringchonse);
    Insnum:=InsStringchonse; 
  END_IF
  IF InsStringchonse>1 THEN
    IntegrationString:= INSERT (IntegrationString,InsOddString,Insnum);	
	   
  END_IF
Insnum:=Insnum+2 ;	
END_FOR

     Stringlen1:= LEN (IntegrationString);

 FOR InsStringlen1:=1 TO (81-Stringlen1) BY 1 DO

      IF InsStringlen1=1 THEN
        stradd:=IntegrationString;
        straddout:=IntegrationString;
        straddout:= INSERT (stradd,' ',Stringlen1);
      END_IF

  straddlen:=Stringlen1+InsStringlen1;
  stradd:=straddout;
  straddout:= INSERT (stradd,' ',straddlen);
    END_FOR


StringTOHmiout:= straddout;//IntegrationString; 
ELSE
//无字符输入处理
IF Stringlen=0 THEN
StringTOHmiout:= MID ('             ',8,5);		
END_IF
//1个字符处理
IF Stringlen=1 THEN
StringTOHmiout:= INSERT (' ',Stringin,1);	
END_IF
END_IF

RStringin:=Stringin;
END_IF

END_FUNCTION_BLOCK
